{attribute 'GeneratedUsingTerminal: EK1122-0000-0018'}
{attribute addProperty BoxType "EK1122-0000-0018"}
{attribute addProperty Id "Beckhoff_ELM3xxx_0030sub_EK1100EK1100_AB5A94672"}
{attribute addProperty CRC "2072767110"}
{attribute addProperty Size "2"}
TYPE Beckhoff_ELM3xxx_0030EK1122_7B8BEA86 EXTENDS EK1122_AB5A9467 :
STRUCT
	{attribute addProperty Name "Beckhoff_ELM3xxx_0030sub_EK1100"}
	{attribute addProperty PreviousPort "Beckhoff ELM3xxx-0030EK1122 : D"}
	Beckhoff_ELM3xxx_0030sub_EK1100 : EK1100_AB5A9467;
END_STRUCT
END_TYPE

(* stored: Version 1.2.0.0, ProductVersion 3.1.4024.9
   DUT Beckhoff_ELM3xxx_0030EK1122_7B8BEA86: Id {18b5382b-389d-467d-aa0b-0906788f7064} *)
